PROGRAM MAIN
VAR
END_VAR

END_PROGRAM

(* stored: Version 1.1.0.1
   POU MAIN: Id {62c77c2f-ebe5-4958-b3da-ed4bf082f032} *)
